// TIA Portal V17 export
// export: Created 2024-08-20T13:37:00.1852425Z, ExportSetting WithDefaults, DisplayName Totally Integrated Automation Portal, DisplayVersion V17 Update 4, DisplayName TIA Portal Openness, DisplayVersion V17 Update 4, DisplayName TIA Portal Version Control Interface, DisplayVersion V17, DisplayName STEP 7 Professional, DisplayVersion V17 Update 4, DisplayName STEP 7 Safety, DisplayVersion V17, DisplayName WinCC Advanced, DisplayVersion V17 Update 4
FUNCTION_BLOCK "MODBUS"   // FB102, LAD
TITLE = BLOCO DE GERENCIAMENTO COMUNICAÇÕES MODBUS/TCP
{ S7_Optimized_Access := 'TRUE' }
VERSION : 0.1
// stored: AutoNumber false, IsIECCheckEnabled false, IsRetainMemResEnabled false, MemoryReserve 100, SetENOAutomatically false, UDAEnableTagReadback false
   VAR
      TEFC0 { S7_SetPoint := 'True'} : TON_TIME;   // Tempo para gerar falha de comunicação
      INI_MOD { S7_SetPoint := 'True'} : TON_TIME;   // Tempo para disparar nova comunicação
      TEFC1 { S7_SetPoint := 'True'} : TON_TIME;   // Tempo para gerar falha de comunicação
      TEFC2 { S7_SetPoint := 'True'} : TON_TIME;   // Tempo para gerar falha de comunicação
      TEFC3 { S7_SetPoint := 'True'} : TON_TIME;   // Tempo para gerar falha de comunicação
      TEFC4 { S7_SetPoint := 'True'} : TON_TIME;   // Tempo para gerar falha de comunicação
      TEFC5 { S7_SetPoint := 'True'} : TON_TIME;   // Tempo para gerar falha de comunicação
      TEFC6 { S7_SetPoint := 'True'} : TON_TIME;   // Tempo para gerar falha de comunicação
      TEFC7 { S7_SetPoint := 'True'} : TON_TIME;   // Tempo para gerar falha de comunicação
      TEFC8 { S7_SetPoint := 'True'} : TON_TIME;   // Tempo para gerar falha de comunicação
      TEFC9 { S7_SetPoint := 'True'} : TON_TIME;   // Tempo para gerar falha de comunicação
      TEFC10 { S7_SetPoint := 'True'} : TON_TIME;   // Tempo para gerar falha de comunicação
      TEFC11 { S7_SetPoint := 'True'} : TON_TIME;   // Tempo para gerar falha de comunicação
      TEFC12 { S7_SetPoint := 'True'} : TON_TIME;   // Tempo para gerar falha de comunicação
      TEFC13 { S7_SetPoint := 'True'} : TON_TIME;   // Tempo para gerar falha de comunicação
      TEFC14 { S7_SetPoint := 'True'} : TON_TIME;   // Tempo para gerar falha de comunicação
      TEFC15 { S7_SetPoint := 'True'} : TON_TIME;   // Tempo para gerar falha de comunicação
      TEFC16 { S7_SetPoint := 'True'} : TON_TIME;   // Tempo para gerar falha de comunicação
      TEFC17 { S7_SetPoint := 'True'} : TON_TIME;   // Tempo para gerar falha de comunicação
      TEFC18 { S7_SetPoint := 'True'} : TON_TIME;   // Tempo para gerar falha de comunicação
      TEFC19 { S7_SetPoint := 'True'} : TON_TIME;   // Tempo para gerar falha de comunicação
      TEFC20 { S7_SetPoint := 'True'} : TON_TIME;   // Tempo para gerar falha de comunicação
      TEFC21 { S7_SetPoint := 'True'} : TON_TIME;   // Tempo para gerar falha de comunicação
      TEFC22 { S7_SetPoint := 'True'} : TON_TIME;   // Tempo para gerar falha de comunicação
      TEFC23 { S7_SetPoint := 'True'} : TON_TIME;   // Tempo para gerar falha de comunicação
      TEFC24 { S7_SetPoint := 'True'} : TON_TIME;   // Tempo para gerar falha de comunicação
      TEFC25 { S7_SetPoint := 'True'} : TON_TIME;   // Tempo para gerar falha de comunicação
      TEFC26 { S7_SetPoint := 'True'} : TON_TIME;   // Tempo para gerar falha de comunicação
      TEFC27 { S7_SetPoint := 'True'} : TON_TIME;   // Tempo para gerar falha de comunicação
      TEFC28 { S7_SetPoint := 'True'} : TON_TIME;   // Tempo para gerar falha de comunicação
   END_VAR
BEGIN

REGION Network 1: INICIA LEITURA MODBUS
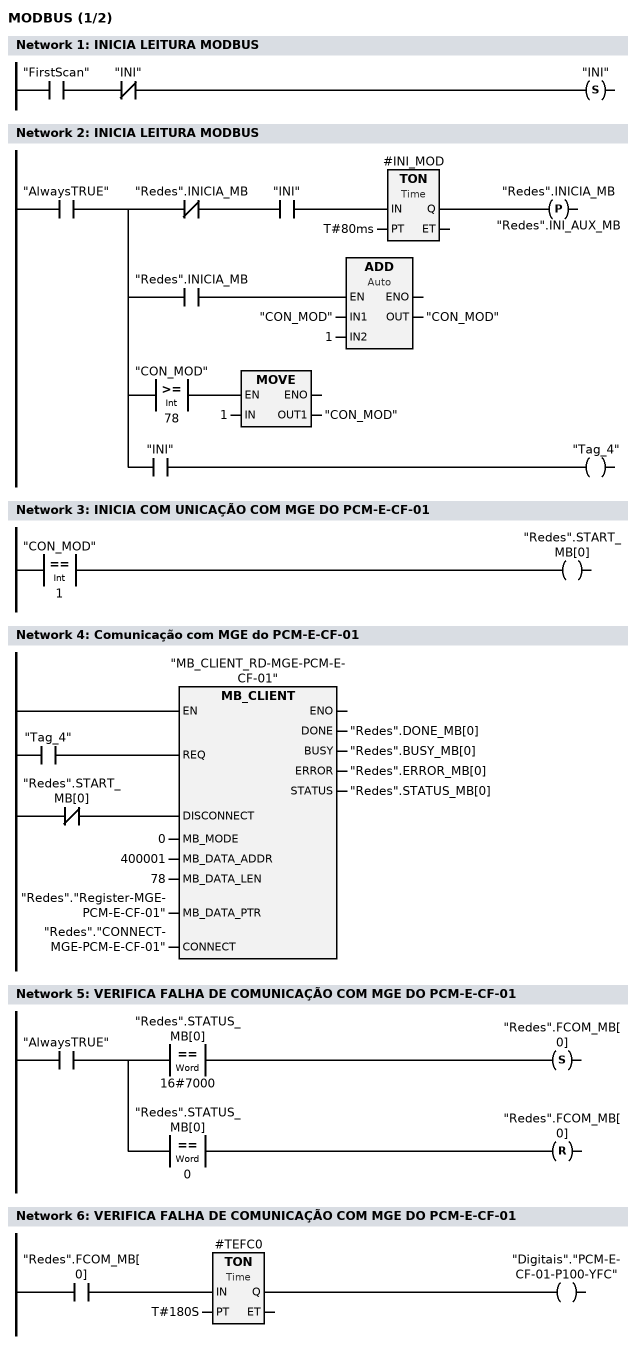
   RUNG wire#powerrail
      Contact( "FirstScan" )
      I_Contact( "INI" )
      S_Coil( "INI" )
   END_RUNG
   // the same network as SCL:
   IF "FirstScan" AND NOT "INI" THEN "INI" := TRUE; END_IF;
END_REGION

REGION Network 2: INICIA LEITURA MODBUS
   #INI_MOD(IN := "AlwaysTRUE" AND NOT "Redes".INICIA_MB AND "INI", PT := T#80ms);   // TON
   "Redes".INICIA_MB := #INI_MOD.Q AND NOT "Redes".INI_AUX_MB;   // rising edge
   "Redes".INI_AUX_MB := #INI_MOD.Q;
   IF "AlwaysTRUE" AND "Redes".INICIA_MB THEN "CON_MOD" := "CON_MOD" + 1; END_IF;
   IF "AlwaysTRUE" AND ("CON_MOD" >= 78) THEN "CON_MOD" := 1; END_IF;
   "Tag_4" := "AlwaysTRUE" AND "INI";
END_REGION

REGION Network 3: INICIA COM UNICAÇÃO COM MGE DO PCM-E-CF-01
   RUNG wire#powerrail
      { S7_Templates := "SrcType := Int" } EQ_Contact(in1 := "CON_MOD", in2 := 1)
      Coil( "Redes".START_MB[0] )
   END_RUNG
   // the same network as SCL:
   "Redes".START_MB[0] := "CON_MOD" = 1;
END_REGION

REGION Network 4: Comunicação com MGE do PCM-E-CF-01
   RUNG wire#powerrail
      "MB_CLIENT_RD-MGE-PCM-E-CF-01".MB_CLIENT(REQ := wire#w1, DISCONNECT := wire#w2, MB_MODE := 0, MB_DATA_ADDR := 400001, MB_DATA_LEN := 78, MB_DATA_PTR := "Redes"."Register-MGE-PCM-E-CF-01", CONNECT := "Redes"."CONNECT-MGE-PCM-E-CF-01", DONE => "Redes".DONE_MB[0], BUSY => "Redes".BUSY_MB[0], ERROR => "Redes".ERROR_MB[0], STATUS => "Redes".STATUS_MB[0])
   END_RUNG
   RUNG wire#powerrail
      Contact( "Tag_4" )
   END_RUNG wire#w1
   RUNG wire#powerrail
      I_Contact( "Redes".START_MB[0] )
   END_RUNG wire#w2
   // the same network as SCL:
   "MB_CLIENT_RD-MGE-PCM-E-CF-01"(REQ := "Tag_4",   // MB_CLIENT
                           DISCONNECT := NOT "Redes".START_MB[0],
                           MB_MODE := 0,
                           MB_DATA_ADDR := 400001,
                           MB_DATA_LEN := 78,
                           MB_DATA_PTR := "Redes"."Register-MGE-PCM-E-CF-01",
                           CONNECT := "Redes"."CONNECT-MGE-PCM-E-CF-01",
                           DONE => "Redes".DONE_MB[0],
                           BUSY => "Redes".BUSY_MB[0],
                           ERROR => "Redes".ERROR_MB[0],
                           STATUS => "Redes".STATUS_MB[0]);
END_REGION

REGION Network 5: VERIFICA FALHA DE COMUNICAÇÃO COM MGE DO PCM-E-CF-01
   RUNG wire#powerrail
      Contact( "AlwaysTRUE" )
      wire#w1
      { S7_Templates := "SrcType := Word" } EQ_Contact(in1 := "Redes".STATUS_MB[0], in2 := 16#7000)
      S_Coil( "Redes".FCOM_MB[0] )
   END_RUNG
   RUNG wire#w1
      { S7_Templates := "SrcType := Word" } EQ_Contact(in1 := "Redes".STATUS_MB[0], in2 := 0)
      R_Coil( "Redes".FCOM_MB[0] )
   END_RUNG
   // the same network as SCL:
   IF "AlwaysTRUE" AND ("Redes".STATUS_MB[0] = 16#7000) THEN "Redes".FCOM_MB[0] := TRUE; END_IF;
   IF "AlwaysTRUE" AND ("Redes".STATUS_MB[0] = 0) THEN "Redes".FCOM_MB[0] := FALSE; END_IF;
END_REGION

REGION Network 6: VERIFICA FALHA DE COMUNICAÇÃO COM MGE DO PCM-E-CF-01
   RUNG wire#powerrail
      Contact( "Redes".FCOM_MB[0] )
      { S7_Templates := "time_type := Time" } #TEFC0.TON(pt := T#180S, et =>)
      Coil( "Digitais"."PCM-E-CF-01-P100-YFC" )
   END_RUNG
   // the same network as SCL:
   #TEFC0(IN := "Redes".FCOM_MB[0], PT := T#180S);   // TON
   "Digitais"."PCM-E-CF-01-P100-YFC" := #TEFC0.Q;
END_REGION

NETWORK
TITLE = Movimentação de dados do MGE PCM-E-CF-01
//CONVERSÃO E MOVIMENTAÇÃO MEDIÇÃO DE TENSÃO
      L     "Redes"."Register-MGE-PCM-E-CF-01"[1];
      DTR;
      L     10.0;
      /R;
      T     "VARIAVEIS"."PCM-E-CF-01-04-P100-ETRS";

      L     "Redes"."Register-MGE-PCM-E-CF-01"[11];
      DTR;
      L     10.0;
      /R;
      T     "VARIAVEIS"."PCM-E-CF-01-04-P100-ETST";

      L     "Redes"."Register-MGE-PCM-E-CF-01"[21];
      DTR;
      L     10.0;
      /R;
      T     "VARIAVEIS"."PCM-E-CF-01-04-P100-ETTR";


//CONVERSÃO E MOVIMENTAÇÃO MEDIÇÃO DE CORRENTE
      L     "Redes"."Register-MGE-PCM-E-CF-01"[2];
      DTR;
      L     100.0;
      /R;
      T     "VARIAVEIS"."PCM-E-CF-01-04-P100-ITR";

      L     "Redes"."Register-MGE-PCM-E-CF-01"[12];
      DTR;
      L     100.0;
      /R;
      T     "VARIAVEIS"."PCM-E-CF-01-04-P100-ITS";

      L     "Redes"."Register-MGE-PCM-E-CF-01"[22];
      DTR;
      L     100.0;
      /R;
      T     "VARIAVEIS"."PCM-E-CF-01-04-P100-ITT";



//CONVERSÃO E MOVIMENTAÇÃO MEDIÇÃO DE POTÊNCIA ATIVA
      L     "Redes"."Register-MGE-PCM-E-CF-01"[34];
      DTR;
      L     100000.0;
      /R;
      T     "VARIAVEIS"."PCM-E-CF-01-04-P100-JPT";

//CONVERSÃO E MOVIMENTAÇÃO MEDIÇÃO DE POTÊNCIA REATIVA
      L     "Redes"."Register-MGE-PCM-E-CF-01"[35];
      DTR;
      L     100000.0;
      /R;
      T     "VARIAVEIS"."PCM-E-CF-01-04-P100-JQT";

//CONVERSÃO E MOVIMENTAÇÃO MEDIÇÃO DE POTÊNCIA APARENTE
      L     "Redes"."Register-MGE-PCM-E-CF-01"[36];
      DTR;
      L     100000.0;
      /R;
      T     "VARIAVEIS"."PCM-E-CF-01-04-P100-JST";

//CONVERSÃO E MOVIMENTAÇÃO MEDIÇÃO DE FATOR DE POTÊNCIA
      L     %DB500.DBW160;
      ITD;
      DTR;
      L     1000.0;
      /R;
      T     "VARIAVEIS"."PCM-E-CF-01-04-P100-FP";



REGION Network 8: INICIA COM UNICAÇÃO COM MGE DO QGBT-AUX-01
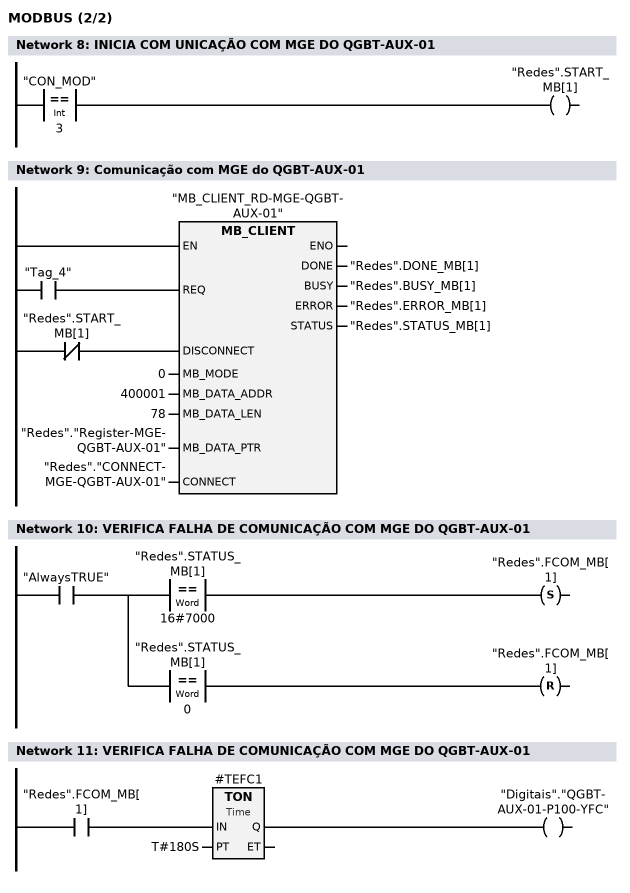
   RUNG wire#powerrail
      { S7_Templates := "SrcType := Int" } EQ_Contact(in1 := "CON_MOD", in2 := 3)
      Coil( "Redes".START_MB[1] )
   END_RUNG
   // the same network as SCL:
   "Redes".START_MB[1] := "CON_MOD" = 3;
END_REGION

REGION Network 9: Comunicação com MGE do QGBT-AUX-01
   RUNG wire#powerrail
      "MB_CLIENT_RD-MGE-QGBT-AUX-01".MB_CLIENT(REQ := wire#w1, DISCONNECT := wire#w2, MB_MODE := 0, MB_DATA_ADDR := 400001, MB_DATA_LEN := 78, MB_DATA_PTR := "Redes"."Register-MGE-QGBT-AUX-01", CONNECT := "Redes"."CONNECT-MGE-QGBT-AUX-01", DONE => "Redes".DONE_MB[1], BUSY => "Redes".BUSY_MB[1], ERROR => "Redes".ERROR_MB[1], STATUS => "Redes".STATUS_MB[1])
   END_RUNG
   RUNG wire#powerrail
      Contact( "Tag_4" )
   END_RUNG wire#w1
   RUNG wire#powerrail
      I_Contact( "Redes".START_MB[1] )
   END_RUNG wire#w2
   // the same network as SCL:
   "MB_CLIENT_RD-MGE-QGBT-AUX-01"(REQ := "Tag_4",   // MB_CLIENT
                           DISCONNECT := NOT "Redes".START_MB[1],
                           MB_MODE := 0,
                           MB_DATA_ADDR := 400001,
                           MB_DATA_LEN := 78,
                           MB_DATA_PTR := "Redes"."Register-MGE-QGBT-AUX-01",
                           CONNECT := "Redes"."CONNECT-MGE-QGBT-AUX-01",
                           DONE => "Redes".DONE_MB[1],
                           BUSY => "Redes".BUSY_MB[1],
                           ERROR => "Redes".ERROR_MB[1],
                           STATUS => "Redes".STATUS_MB[1]);
END_REGION

REGION Network 10: VERIFICA FALHA DE COMUNICAÇÃO COM MGE DO QGBT-AUX-01
   RUNG wire#powerrail
      Contact( "AlwaysTRUE" )
      wire#w1
      { S7_Templates := "SrcType := Word" } EQ_Contact(in1 := "Redes".STATUS_MB[1], in2 := 16#7000)
      S_Coil( "Redes".FCOM_MB[1] )
   END_RUNG
   RUNG wire#w1
      { S7_Templates := "SrcType := Word" } EQ_Contact(in1 := "Redes".STATUS_MB[1], in2 := 0)
      R_Coil( "Redes".FCOM_MB[1] )
   END_RUNG
   // the same network as SCL:
   IF "AlwaysTRUE" AND ("Redes".STATUS_MB[1] = 16#7000) THEN "Redes".FCOM_MB[1] := TRUE; END_IF;
   IF "AlwaysTRUE" AND ("Redes".STATUS_MB[1] = 0) THEN "Redes".FCOM_MB[1] := FALSE; END_IF;
END_REGION

REGION Network 11: VERIFICA FALHA DE COMUNICAÇÃO COM MGE DO QGBT-AUX-01
   RUNG wire#powerrail
      Contact( "Redes".FCOM_MB[1] )
      { S7_Templates := "time_type := Time" } #TEFC1.TON(pt := T#180S, et =>)
      Coil( "Digitais"."QGBT-AUX-01-P100-YFC" )
   END_RUNG
   // the same network as SCL:
   #TEFC1(IN := "Redes".FCOM_MB[1], PT := T#180S);   // TON
   "Digitais"."QGBT-AUX-01-P100-YFC" := #TEFC1.Q;
END_REGION

NETWORK
TITLE = Movimentação de dados do MGE QGBT-AUX-01
//CONVERSÃO E MOVIMENTAÇÃO MEDIÇÃO DE TENSÃO
      L     "Redes"."Register-MGE-QGBT-AUX-01"[1];
      DTR;
      L     10.0;
      /R;
      T     "VARIAVEIS"."QGBT-AUX-01-P100-ETRS";

      L     "Redes"."Register-MGE-QGBT-AUX-01"[11];
      DTR;
      L     10.0;
      /R;
      T     "VARIAVEIS"."QGBT-AUX-01-P100-ETST";

      L     "Redes"."Register-MGE-QGBT-AUX-01"[21];
      DTR;
      L     10.0;
      /R;
      T     "VARIAVEIS"."QGBT-AUX-01-P100-ETTR";


//CONVERSÃO E MOVIMENTAÇÃO MEDIÇÃO DE CORRENTE
      L     "Redes"."Register-MGE-QGBT-AUX-01"[2];
      DTR;
      L     100.0;
      /R;
      T     "VARIAVEIS"."QGBT-AUX-01-P100-ITR";

      L     "Redes"."Register-MGE-QGBT-AUX-01"[12];
      DTR;
      L     100.0;
      /R;
      T     "VARIAVEIS"."QGBT-AUX-01-P100-ITS";

      L     "Redes"."Register-MGE-QGBT-AUX-01"[22];
      DTR;
      L     100.0;
      /R;
      T     "VARIAVEIS"."QGBT-AUX-01-P100-ITT";



//CONVERSÃO E MOVIMENTAÇÃO MEDIÇÃO DE POTÊNCIA ATIVA
      L     "Redes"."Register-MGE-QGBT-AUX-01"[34];
      DTR;
      L     100000.0;
      /R;
      T     "VARIAVEIS"."QGBT-AUX-01-P100-JPT";

//CONVERSÃO E MOVIMENTAÇÃO MEDIÇÃO DE POTÊNCIA REATIVA
      L     "Redes"."Register-MGE-QGBT-AUX-01"[35];
      DTR;
      L     100000.0;
      /R;
      T     "VARIAVEIS"."QGBT-AUX-01-P100-JQT";

//CONVERSÃO E MOVIMENTAÇÃO MEDIÇÃO DE POTÊNCIA APARENTE
      L     "Redes"."Register-MGE-QGBT-AUX-01"[36];
      DTR;
      L     100000.0;
      /R;
      T     "VARIAVEIS"."QGBT-AUX-01-P100-JST";

//CONVERSÃO E MOVIMENTAÇÃO MEDIÇÃO DE FATOR DE POTÊNCIA
      L     %DB500.DBW316;
      ITD;
      DTR;
      L     1000.0;
      /R;
      T     "VARIAVEIS"."QGBT-AUX-01-P100-FP";


END_FUNCTION_BLOCK
